// TwinCAT 3 PLC project Flyweight
// ProgramVersion: 3.1.4023.0
// libraries:
//   Tc2_Standard, * (Beckhoff Automation GmbH)
//   Tc2_System, * (Beckhoff Automation GmbH)
//   Tc3_Module, * (Beckhoff Automation GmbH)
// project tree:
//   / Class Diagram.TcCD (not stored), Param.TcGVL, PlcTask.TcTTO
//   Classes/ Car.TcPOU, FlyweightFactory.TcPOU
//   ITFs/ I_Car.TcIO
//   POUs/ MAIN.TcPOU
// real-time tasks:
//   TASK PlcTask: cycle T#10ms, priority 20, ADS port 350

CONFIGURATION Flyweight
    RESOURCE PLC ON TwinCAT3
        TASK PlcTask(INTERVAL := T#10ms, PRIORITY := 20);
        PROGRAM MAIN WITH PlcTask : MAIN;
    END_RESOURCE
END_CONFIGURATION

// ---- Param.TcGVL
{attribute 'qualified_only'}
VAR_GLOBAL CONSTANT
	iMaxArray : INT := 5;
END_VAR

// ---- ITFs/I_Car.TcIO
INTERFACE I_Car

METHOD PUBLIC ShowDetails : STRING
END_METHOD

END_INTERFACE

// ---- POUs/MAIN.TcPOU
PROGRAM MAIN
VAR
	Colors 		: ARRAY [1..Param.iMaxArray] OF STRING  := ['black', 'white', 'blue', 'green', 'brown' ];
	Patents 	: ARRAY [1..Param.iMaxArray] OF STRING  := ['patent11', 'patent22', 'patent33', 'patent44', 'patent55'];
	Owners 		: ARRAY [1..Param.iMaxArray] OF STRING  := ['Victor', 'Jesus', 'Alex', 'Hugo', 'David'];
	
	flyweightFactory : FlyweightFactory;
	
	bExecute : BOOL;
		
END_VAR


IF bExecute THEN
	
	flyweightFactory.ListCars(Colors, Patents, Owners);
	
	bExecute := FALSE;
	
END_IF

END_PROGRAM

// ---- Classes/FlyweightFactory.TcPOU
FUNCTION_BLOCK PUBLIC FlyweightFactory
VAR
	pCar : POINTER TO Car;
END_VAR


METHOD FB_exit : BOOL
VAR_INPUT
	bInCopyCode : BOOL; // if TRUE, the exit method is called for exiting an instance that is copied afterwards (online change).
END_VAR
VAR
	i : INT;
END_VAR

//FOR i := 1 TO Param.iMaxArray BY 1 DO
	
	IF (pCar <> 0) THEN
		
    	__DELETE(pCar);
 
	END_IF
	
//END_FOR
END_METHOD


METHOD PUBLIC ListCars
VAR_INPUT
	Color 	: ARRAY [1..Param.iMaxArray] OF STRING;
	Patent 	: ARRAY [1..Param.iMaxArray] OF STRING;
	Owner 	: ARRAY [1..Param.iMaxArray] OF STRING;
END_VAR
VAR
	i : INT;
END_VAR

IF (pCar = 0) THEN
				
	pCar := __NEW(Car);
	
END_IF		

FOR i := 1 TO Param.iMaxArray BY 1 DO
	
//	IF (pVehicle = 0) THEN
				
//		pVehicle := __NEW(Auto);
		
		pCar^.setColor(Color[i]);

		pCar^.setPatent(Patent[i]);	

		pCar^.setOwner(Owner[i]);				
		
 		ADSLOGSTR( msgCtrlMask := ADSLOG_MSGTYPE_HINT, msgFmtStr := 'Data Car: %s', strArg := pCar^.ShowDetails());
		
//		IF (pVehicle <> 0) THEN
		
//    		__DELETE(pVehicle);
 
//		END_IF
		
//	END_IF
	
END_FOR
END_METHOD

END_FUNCTION_BLOCK

// ---- Classes/Car.TcPOU
{attribute 'enable_dynamic_creation'}
FUNCTION_BLOCK Car IMPLEMENTS I_Car
VAR
	_Color : STRING;
	_Patent : STRING;
	_Owner : STRING;
END_VAR

METHOD setColor
VAR_INPUT
	Color : STRING;
END_VAR
THIS^._Color := Color;
END_METHOD

METHOD setOwner
VAR_INPUT
	Owner : STRING;
END_VAR
 THIS^._Owner := Owner;
END_METHOD

METHOD setPatent
VAR_INPUT
	Patent : STRING;
END_VAR
THIS^._Patent := Patent;
END_METHOD


METHOD ShowDetails : STRING
VAR
	sPatent : STRING;
	sColor	: STRING;
	sOwner	: STRING;
END_VAR

sPatent := CONCAT(STR1:='Patent: ' , STR2:= THIS^._Patent);
sColor 	:= CONCAT(STR1:=', Color: ' , STR2:= THIS^._Color);
sOwner 	:= CONCAT(STR1:=', Owner: ' , STR2:= THIS^._Owner);

ShowDetails := CONCAT(STR1:= sPatent , STR2:= CONCAT(STR1:= sColor , STR2:= sOwner));
END_METHOD

END_FUNCTION_BLOCK
